INTERFACE ITF_GroupE_TE2 EXTENDS ITF_BaseGroupElement

METHOD testMethodGE : BOOL
VAR_INPUT
END_VAR
END_METHOD

END_INTERFACE

(* stored: Version 1.1.0.1, ProductVersion 3.1.4024.15
   Itf ITF_GroupE_TE2: Id {ee118838-fbb2-4bcc-866c-d67c7c70751e}
   Method testMethodGE: Id {58d6bc74-7fdb-4186-b5f3-2b34c14c2343} *)
